TYPE st_ModbusSwitchOff :
STRUCT
	switchOff_1 : BOOL :=FALSE;
	switchOff_2 : BOOL :=FALSE;
	switchOff_3 : BOOL :=FALSE;
	switchOff_4 : BOOL :=FALSE;
END_STRUCT
END_TYPE

(* stored: Version 1.1.0.1, ProductVersion 3.1.4024.13
   DUT st_ModbusSwitchOff: Id {f172d03a-f5e5-4455-891f-c4b0bda3f17d} *)
